KUKA KRL program: Lequn_Singlebead_powder.src, Lequn_Singlebead_powder.dat

--- Lequn_Singlebead_powder.src ---
&ACCESS RVO
&REL 231
&PARAM DISKPATH = KRC:\R1\Program\Lequn
DEF Lequn_Singlebead_powder( )

 DECL E6POS LayerStartPt
 DECL E6POS LayerStartPt2
   DECL E6POS XP2
   DECL E6POS XP3
   DECL E6POS XP4
   DECL REAL stepover
   DECL REAL stepover1 ; step over between contour and infill
   DECL REAL xLength
   DECL REAL yWidth
   DECL REAL layerHt
   DECL INT YSTEP
   DECL INT YSTEP_MAX
   DECL INT XSTEP
   DECL INT XSTEP_MAX
   DECL INT nLayers ;  the total number of layers
   DECL INT layer ; the current layer number
   DECL REAL power
   DECL INT count;
   DECL REAL B_angle; laser tilt in degree
   DECL REAL C_angle; laser tilt in degree
   DECL FRAME relpos


   ;---------------------RSI variable--------------------
   ; Declaration of KRL variables
   DECL INT ret	; Return value for RSI commands
   DECL INT CONTID	; ContainerID
   ;---------------------RSI variable--------------------

   ;---------------------RSI --------------------
   ret = RSI_CREATE("ros_rsi",CONTID,TRUE)
   IF (ret <> RSIOK) THEN
      HALT
   ENDIF

   ; Start RSI execution
   ret = RSI_ON(#ABSOLUTE)
   IF (ret <> RSIOK) THEN
      HALT
   ENDIF
   ;---------------------RSI--------------------


         GLOBAL INTERRUPT DECL 3 WHEN $STOPMESS==TRUE DO IR_STOPM ( )
         INTERRUPT ON 3
         BAS (#INITMOV,0 )

   ptp $POS_ACT
   ;FOLD LIN P1 Vel=0.02 m/s CPDAT1 Tool[1]:LASER Base[0] ;%{PE}
;FOLD Parameters ;%{h}
;Params IlfProvider=kukaroboter.basistech.inlineforms.movement.old; Kuka.IsGlobalPoint=False; Kuka.PointName=P1; Kuka.BlendingEnabled=False; Kuka.MoveDataName=CPDAT1; Kuka.VelocityPath=0.02; Kuka.CurrentCDSetIndex=0; Kuka.MovementParameterFieldEnabled=True; IlfCommand=LIN
;ENDFOLD

$BWDSTART = FALSE
LDAT_ACT = LCPDAT1
FDAT_ACT = FP1
BAS(#CP_PARAMS, 0.02)
SET_CD_PARAMS (0)
LIN XP1
;ENDFOLD




   ;--------------Process variables-----------------
   stepover = 2.0 ;mm
   xLength = 90.0 ;mm
   ;yWidth = 70.0 ;mm
   layerHt = 0.4 ;mm
   nLayers = 50
   ;B_angle = 25 ; tilt @ 25 degree
   ;C_angle =25 ; degree
   $VEL.CP=0.0275 ; SPEED in m/s
   $APO.CDIS = 0.2 ; mm ; equivalent to Zone data in ABB (Z0)
   $ANOUT[1]=0.219 ; laser power in voltage
   ;$ANOUT[2]=0.2125 ; wire feed rate in voltage
   ;-------------------------------------------------

   relpos = {X 0, Y 0, Z 0, A 0, B 0, C 0}

   $OUT[15]=TRUE ; Wire touch signal bypass

   LIN XP1
   LaserOn_Ext() ; on laser

   count = 1

   For layer = 1 TO nLayers STEP 1
      IF(layer/2) <>(layer/2.0) THEN
         ; move to start point
         LayerStartPt = XP1
         LayerStartPt.z = XP1.Z + layerHt * (layer - 1)
         LIN LayerStartPt
         ;odd layer


         LaserStart_Ext()

         relpos = {X 0, Y 0, Z 0, A 0, B 0, C 0}
         relpos.X = xLength
         LIN_REL relpos


         LaserEnd_Ext()
         WAIT SEC 5.0
         count = count +1




      Else
         ;even layer
         ; move to start point
         LayerStartPt = XP1
         LayerStartPt.z = XP1.Z + layerHt * (layer - 1)
         LayerStartPt.x = XP1.x + xLength
         LIN LayerStartPt


         LaserStart_Ext()

         relpos = {X 0, Y 0, Z 0, A 0, B 0, C 0}
         relpos.X = -xLength
         LIN_REL relpos

         LaserEnd_Ext()


         WAIT SEC 5.0
         count = count +1




       ENDIF
         LaserEnd_Ext()

   ENDFOR
   LaserOff_Ext()
   WAIT SEC 2.0

END

--- Lequn_Singlebead_powder.dat ---
&ACCESS RVO
&REL 231
&PARAM DISKPATH = KRC:\R1\Program\Lequn
DEFDAT  LEQUN_SINGLEBEAD_POWDER
;FOLD EXTERNAL DECLARATIONS;%{PE}%MKUKATPBASIS,%CEXT,%VCOMMON,%P
;FOLD BASISTECH EXT;%{PE}%MKUKATPBASIS,%CEXT,%VEXT,%P
EXT  BAS (BAS_COMMAND  :IN,REAL  :IN )
DECL INT SUCCESS
;ENDFOLD (BASISTECH EXT)
;FOLD USER EXT;%{E}%MKUKATPUSER,%CEXT,%VEXT,%P
;Make your modifications here

;ENDFOLD (USER EXT)
;ENDFOLD (EXTERNAL DECLARATIONS)
DECL E6POS XP1={X 2983.45361,Y -1764.81641,Z 918.625366,A -90.1096497,B -0.521237314,C 178.019348,S 22,T 51,E1 -1324.94714,E2 0.00743009709,E3 -0.715414524,E4 0.0,E5 0.0,E6 0.0}
DECL FDAT FP1={TOOL_NO 1,BASE_NO 0,IPO_FRAME #BASE,POINT2[] " "}
DECL LDAT LCPDAT1={VEL 0.0200000,ACC 100.000,APO_DIST 500.000,APO_FAC 50.0000,AXIS_VEL 100.000,AXIS_ACC 100.000,ORI_TYP #VAR,CIRC_TYP #BASE,JERK_FAC 50.0000,GEAR_JERK 100.000,EXAX_IGN 0}
DECL MODULEPARAM_T LAST_TP_PARAMS={PARAMS[] "Kuka.PointName=P1; Kuka.FrameData.base_no=0; Kuka.FrameData.tool_no=1; Kuka.FrameData.ipo_frame=#BASE; Kuka.isglobalpoint=False; Kuka.MoveDataName=CPDAT1; Kuka.MovementData.apo_fac=50; Kuka.MovementData.apo_dist=500; Kuka.MovementData.axis_acc=100; Kuka.MovementData.axis_vel=100; Kuka.MovementData.circ_typ=#BASE; Kuka.MovementData.jerk_fac=50; Kuka.MovementData.ori_typ=#VAR; Kuka.MovementData.vel=0.02; Kuka.MovementData.acc=100; Kuka.MovementData.exax_ign=0; Kuka.VelocityPath=0.02; Kuka.BlendingEnabled=False; Kuka.CurrentCDSetIndex=0; SyncLabel=AutoSync; Kuka.FrameData.point2=      "}
DECL E6POS XP5={X 1267.51770,Y -1547.66406,Z 1189.19409,A -89.9841156,B -0.616697371,C 178.079834,S 22,T 51,E1 -1150.03894,E2 0.00427939091,E3 -1.87918558E-05,E4 0.0,E5 0.0,E6 0.0}
DECL E6POS XP6={X 2336.54956,Y -1328.21008,Z 942.745,A -89.9947586,B -0.533553302,C 177.973938,S 22,T 51,E1 -1149.45276,E2 0.00158752210,E3 -3.00910284E-14,E4 0.0,E5 0.0,E6 0.0}
DECL E6POS XP7={X 3009.99805,Y -1744.91968,Z 1023.21338,A 0.000410029199,B -0.407568067,C 179.281097,S 22,T 51,E1 -1318.66443,E2 0.00737420097,E3 -1.81965232,E4 0.0,E5 0.0,E6 0.0}
ENDDAT
